(* IEC 61131-3 sources: sphere-usecases/sector-water/rovisys-distribution/implementations/openplc/st, 2 files *)

(* ---- wd_controller.st ---- *)
(*
 * Water Distribution UC0 Controller
 * SPHERE CPS Enclave - OpenPLC Implementation
 *
 * IEC 61131-3 Structured Text (OpenPLC/matiec compatible)
 *
 * This controller manages:
 *   - Supply Line: Supply tank level control, pump operation
 *   - Distribution Grid: Elevated tank filling via valve control
 *   - Return Water System: RWS tank level control, pump operation
 *
 * Architecture:
 *   Controller PLC <-> Modbus Bridge <-> Simulator PLC
 *
 * I/O Mapping (configured in OpenPLC web interface):
 *   Inputs from Simulator (via Bridge):
 *     ai_supply_tank_level -> %IW70
 *     ai_supply_pump_flow -> %IW71
 *     ai_supply_naocl_level -> %IW72
 *     ai_supply_nh4cl_level -> %IW73
 *     ai_grid_elev_level -> %IW74
 *     ai_grid_consum_level -> %IW75
 *     ai_rws_tank_level -> %IW76
 *     di_supply_pump_sts -> %IX2.0
 *     di_supply_mixer_sts -> %IX2.1
 *     di_supply_valve_sts -> %IX2.2
 *     di_grid_elev_valve_sts -> %IX2.3
 *     di_rws_pump_sts -> %IX2.4
 *     di_rws_valve_sts -> %IX2.5
 *     hmi_start -> %IX0.0
 *     hmi_stop -> %IX0.1
 *
 *   Outputs to Simulator (via Bridge):
 *     ao_supply_pump_speed -> %QW100
 *     ao_rws_pump_speed -> %QW101
 *     do_supply_valve -> %QX5.0
 *     do_grid_elev_valve -> %QX5.1
 *     do_rws_valve -> %QX5.2
 *     do_sys_idle -> %QX7.0
 *     do_sys_running -> %QX7.1
 *     do_alarm_supply_hh -> %QX8.0
 *)

(* System State Type - Using INT since iec2c doesn't support ENUM well *)
(* 0=IDLE, 1=START, 2=RUNNING, 3=SHUTDOWN *)

PROGRAM MainProgram
  VAR_INPUT
    (* Analog Inputs from Simulator *)
    ai_supply_tank_level : REAL;      (* Supply tank level [mm] *)
    ai_supply_pump_flow : REAL;       (* Supply pump flow [L/min] *)
    ai_supply_naocl_level : REAL;     (* NaOCl tank level [mm] *)
    ai_supply_nh4cl_level : REAL;     (* NH4Cl tank level [mm] *)
    ai_grid_elev_level : REAL;        (* Elevated tank level [mm] *)
    ai_grid_consum_level : REAL;      (* Consumer tank level [mm] *)
    ai_rws_tank_level : REAL;         (* RWS tank level [mm] *)

    (* Digital Inputs from Simulator *)
    di_supply_pump_sts : BOOL;        (* Supply pump running *)
    di_supply_mixer_sts : BOOL;       (* Supply mixer running *)
    di_supply_valve_sts : BOOL;       (* Supply valve open *)
    di_grid_elev_valve_sts : BOOL;    (* Elevated tank valve open *)
    di_rws_pump_sts : BOOL;           (* RWS pump running *)
    di_rws_valve_sts : BOOL;          (* RWS valve open *)

    (* HMI Inputs *)
    hmi_start : BOOL;                 (* Start button *)
    hmi_stop : BOOL;                  (* Stop button *)
  END_VAR

  VAR_OUTPUT
    (* Analog Outputs to Simulator *)
    ao_supply_pump_speed : REAL;      (* Supply pump speed [%] *)
    ao_rws_pump_speed : REAL;         (* RWS pump speed [%] *)

    (* Digital Outputs to Simulator *)
    do_supply_valve : BOOL;           (* Supply valve command *)
    do_grid_elev_valve : BOOL;        (* Elevated tank valve command *)
    do_rws_valve : BOOL;              (* RWS valve command *)

    (* System State Outputs *)
    do_sys_idle : BOOL;               (* System idle state *)
    do_sys_running : BOOL;            (* System running state *)

    (* Alarm Outputs *)
    do_alarm_supply_hh : BOOL;        (* Supply tank HH alarm *)
  END_VAR

  VAR
    (* System State Machine - 0=IDLE, 1=START, 2=RUNNING, 3=SHUTDOWN *)
    sys_state : INT := 0;
    permissive_supply_ok : BOOL := FALSE;
    permissive_grid_ok : BOOL := FALSE;
    permissives_ready : BOOL := FALSE;

    (* Control Setpoints *)
    supply_tank_low_sp : REAL := 500.0;         (* Start pump below this [mm] *)
    supply_tank_high_sp : REAL := 1200.0;       (* Stop pump above this [mm] *)
    supply_tank_hh_sp : REAL := 1200.0;         (* HH alarm threshold [mm] *)

    grid_elev_low_sp : REAL := 600.0;           (* Open valve below this [mm] *)
    grid_elev_high_sp : REAL := 1600.0;         (* Close valve above this [mm] *)

    rws_tank_low_sp : REAL := 300.0;            (* Start pump below this [mm] *)
    rws_tank_high_sp : REAL := 1200.0;          (* Stop pump above this [mm] *)

    (* Pump Speed Setpoints *)
    supply_pump_normal_speed : REAL := 75.0;    (* Normal operating speed [%] *)
    rws_pump_normal_speed : REAL := 50.0;       (* Normal operating speed [%] *)

    (* Internal State *)
    supply_pump_cmd : BOOL := FALSE;
    rws_pump_cmd : BOOL := FALSE;
  END_VAR

  (* State constants *)
  (* STATE_IDLE = 0; STATE_START = 1; STATE_RUNNING = 2; STATE_SHUTDOWN = 3 *)

  CASE sys_state OF

    0: (* STATE_IDLE - System is idle, waiting for start command *)
      do_sys_idle := TRUE;
      do_sys_running := FALSE;

      (* All outputs off in idle *)
      ao_supply_pump_speed := 0.0;
      ao_rws_pump_speed := 0.0;
      do_supply_valve := FALSE;
      do_grid_elev_valve := FALSE;
      do_rws_valve := FALSE;

      (* Transition: Start button pressed *)
      IF hmi_start AND NOT hmi_stop THEN
        sys_state := 1;
      END_IF;

    1: (* STATE_START - Starting up, check permissives *)
      do_sys_idle := FALSE;
      do_sys_running := FALSE;

      (* Check permissives *)
      permissive_supply_ok := (ai_supply_tank_level > 300.0);
      permissive_grid_ok := (ai_grid_elev_level < 5500.0);
      permissives_ready := permissive_supply_ok AND permissive_grid_ok;

      (* Transition: Permissives met -> RUNNING *)
      IF permissives_ready THEN
        sys_state := 2;
      END_IF;

      (* Transition: Stop pressed -> SHUTDOWN *)
      IF hmi_stop THEN
        sys_state := 3;
      END_IF;

    2: (* STATE_RUNNING - Normal operation *)
      do_sys_idle := FALSE;
      do_sys_running := TRUE;

      (* SUPPLY LINE CONTROL *)
      (* Level-based pump control *)
      IF ai_supply_tank_level <= supply_tank_low_sp THEN
        supply_pump_cmd := TRUE;
      ELSIF ai_supply_tank_level >= supply_tank_high_sp THEN
        supply_pump_cmd := FALSE;
      END_IF;

      (* Set pump speed *)
      IF supply_pump_cmd THEN
        ao_supply_pump_speed := supply_pump_normal_speed;
        do_supply_valve := TRUE;
      ELSE
        ao_supply_pump_speed := 0.0;
        do_supply_valve := FALSE;
      END_IF;

      (* Supply tank HH alarm *)
      IF ai_supply_tank_level >= supply_tank_hh_sp THEN
        do_alarm_supply_hh := TRUE;
      ELSE
        do_alarm_supply_hh := FALSE;
      END_IF;

      (* DISTRIBUTION GRID CONTROL *)
      IF ai_grid_elev_level <= grid_elev_low_sp THEN
        do_grid_elev_valve := TRUE;
      ELSIF ai_grid_elev_level >= grid_elev_high_sp THEN
        do_grid_elev_valve := FALSE;
      END_IF;

      (* RETURN WATER SYSTEM CONTROL *)
      IF ai_rws_tank_level >= rws_tank_high_sp THEN
        rws_pump_cmd := TRUE;
      ELSIF ai_rws_tank_level <= rws_tank_low_sp THEN
        rws_pump_cmd := FALSE;
      END_IF;

      IF rws_pump_cmd THEN
        ao_rws_pump_speed := rws_pump_normal_speed;
        do_rws_valve := TRUE;
      ELSE
        ao_rws_pump_speed := 0.0;
        do_rws_valve := FALSE;
      END_IF;

      (* Transition: Stop pressed -> SHUTDOWN *)
      IF hmi_stop THEN
        sys_state := 3;
      END_IF;

    3: (* STATE_SHUTDOWN - Shutting down *)
      do_sys_idle := FALSE;
      do_sys_running := FALSE;

      (* Stop all pumps *)
      ao_supply_pump_speed := 0.0;
      ao_rws_pump_speed := 0.0;
      supply_pump_cmd := FALSE;
      rws_pump_cmd := FALSE;

      (* Close all valves *)
      do_supply_valve := FALSE;
      do_grid_elev_valve := FALSE;
      do_rws_valve := FALSE;

      (* Clear alarms *)
      do_alarm_supply_hh := FALSE;

      (* Clear permissives *)
      permissive_supply_ok := FALSE;
      permissive_grid_ok := FALSE;
      permissives_ready := FALSE;

      (* Transition: Stop released -> IDLE *)
      IF NOT hmi_stop THEN
        sys_state := 0;
      END_IF;

  END_CASE;

END_PROGRAM

(* ---- wd_simulator.st ---- *)
(*
 * Water Distribution UC0 Simulator
 * SPHERE CPS Enclave - OpenPLC Implementation
 *
 * IEC 61131-3 Structured Text (OpenPLC/matiec compatible)
 *
 * This simulator models the physical dynamics of:
 *   - Supply Line: Supply tank, chemical tanks, pump, valves
 *   - Distribution Grid: Elevated tank, consumer tank, valves
 *   - Return Water System: RWS tank, pump, valves
 *
 * Architecture:
 *   Controller PLC <-> Modbus Bridge <-> Simulator PLC (this)
 *
 * I/O Mapping (configured in OpenPLC web interface):
 *   Command Inputs (from Controller via Bridge):
 *     cmd_supply_pump_speed -> %QW200
 *     cmd_rws_pump_speed -> %QW201
 *     cmd_supply_valve -> %QX3.0
 *     cmd_grid_elev_valve -> %QX3.1
 *     cmd_rws_valve -> %QX3.2
 *
 *   Sensor Outputs (to Controller via Bridge):
 *     out_supply_tank_level -> %QW300
 *     out_supply_pump_flow -> %QW301
 *     out_supply_naocl_level -> %QW302
 *     out_supply_nh4cl_level -> %QW303
 *     out_grid_elev_level -> %QW304
 *     out_grid_consum_level -> %QW305
 *     out_rws_tank_level -> %QW306
 *
 *   Status Outputs (to Controller via Bridge):
 *     out_supply_pump_sts -> %QX40.0
 *     out_supply_mixer_sts -> %QX40.1
 *     out_supply_valve_sts -> %QX40.2
 *     out_grid_elev_valve_sts -> %QX40.3
 *     out_rws_pump_sts -> %QX40.4
 *     out_rws_valve_sts -> %QX40.5
 *)

PROGRAM MainProgram
  VAR_INPUT
    (* Command Inputs from Controller via Bridge *)
    cmd_supply_pump_speed : REAL;     (* Supply pump speed cmd [%] *)
    cmd_rws_pump_speed : REAL;        (* RWS pump speed cmd [%] *)
    cmd_supply_valve : BOOL;          (* Supply valve command *)
    cmd_grid_elev_valve : BOOL;       (* Elevated tank valve cmd *)
    cmd_rws_valve : BOOL;             (* RWS valve command *)
  END_VAR

  VAR_OUTPUT
    (* Sensor Outputs to Controller via Bridge *)
    out_supply_tank_level : REAL;     (* Supply tank level [mm] *)
    out_supply_pump_flow : REAL;      (* Supply pump flow [L/min] *)
    out_supply_naocl_level : REAL;    (* NaOCl tank level [mm] *)
    out_supply_nh4cl_level : REAL;    (* NH4Cl tank level [mm] *)
    out_grid_elev_level : REAL;       (* Elevated tank level [mm] *)
    out_grid_consum_level : REAL;     (* Consumer tank level [mm] *)
    out_rws_tank_level : REAL;        (* RWS tank level [mm] *)

    (* Status Outputs to Controller via Bridge *)
    out_supply_pump_sts : BOOL;       (* Supply pump running *)
    out_supply_mixer_sts : BOOL;      (* Supply mixer running *)
    out_supply_valve_sts : BOOL;      (* Supply valve open *)
    out_grid_elev_valve_sts : BOOL;   (* Elevated tank valve open *)
    out_rws_pump_sts : BOOL;          (* RWS pump running *)
    out_rws_valve_sts : BOOL;         (* RWS valve open *)
  END_VAR

  VAR
    (* Simulation Constants - Timing *)
    DT_SEC : REAL := 0.1;                       (* Simulation timestep [s] *)
    MOTORIZED_VALVE_DELAY : INT := 600;         (* 60s at 100ms scan *)
    PUMP_SPINUP_DELAY : INT := 20;              (* 2s at 100ms scan *)

    (* Physical parameters - Supply *)
    SUPPLY_TANK_AREA_M2 : REAL := 40.0;
    SUPPLY_TANK_MAX_MM : REAL := 1500.0;
    SUPPLY_INFLOW_LPM : REAL := 150.0;
    SUPPLY_PUMP_MAX_LPM : REAL := 200.0;

    (* Physical parameters - Chemical tanks *)
    NAOCL_TANK_AREA_M2 : REAL := 0.1;
    NAOCL_DOSE_LPM : REAL := 0.038;
    NH4CL_TANK_AREA_M2 : REAL := 0.1;
    NH4CL_DOSE_LPM : REAL := 0.019;

    (* Physical parameters - Grid *)
    ELEV_TANK_AREA_M2 : REAL := 60.0;
    ELEV_TANK_MAX_MM : REAL := 2000.0;
    CONSUM_TANK_AREA_M2 : REAL := 10.0;
    CONSUM_TANK_MAX_MM : REAL := 2000.0;
    GRID_DEMAND_LPM : REAL := 100.0;
    ELEV_DRAIN_LPM : REAL := 300.0;

    (* Physical parameters - RWS *)
    RWS_TANK_AREA_M2 : REAL := 0.3;
    RWS_TANK_MAX_MM : REAL := 1500.0;
    RWS_PUMP_MAX_LPM : REAL := 38.0;
    RETURN_FRACTION : REAL := 0.9;

    (* Tank levels [mm] *)
    supply_tank_level : REAL := 1000.0;
    naocl_tank_level : REAL := 800.0;
    nh4cl_tank_level : REAL := 800.0;
    grid_elev_level : REAL := 1200.0;
    grid_consum_level : REAL := 1000.0;
    rws_tank_level : REAL := 500.0;

    (* Valve states with delay modeling *)
    supply_valve_timer : INT := 0;
    supply_valve_state : BOOL := FALSE;
    grid_elev_valve_timer : INT := 0;
    grid_elev_valve_state : BOOL := FALSE;
    rws_valve_timer : INT := 0;
    rws_valve_state : BOOL := FALSE;

    (* Pump states with delay modeling *)
    supply_pump_timer : INT := 0;
    supply_pump_state : BOOL := FALSE;
    supply_pump_actual_speed : REAL := 0.0;
    rws_pump_timer : INT := 0;
    rws_pump_state : BOOL := FALSE;
    rws_pump_actual_speed : REAL := 0.0;

    (* Flow rates [L/min] *)
    supply_pump_flow : REAL := 0.0;
    rws_pump_flow : REAL := 0.0;
    grid_demand_actual : REAL := 0.0;
    return_flow : REAL := 0.0;

    (* Mixer state *)
    mixer_running : BOOL := TRUE;

    (* Temporary calculation variables *)
    delta_level : REAL := 0.0;
    flow_in : REAL := 0.0;
    flow_out : REAL := 0.0;
  END_VAR

  (* =====================================================================
     VALVE DELAY MODELING
     ===================================================================== *)

  (* Supply Tank Valve *)
  IF cmd_supply_valve AND NOT supply_valve_state THEN
    supply_valve_timer := supply_valve_timer + 1;
    IF supply_valve_timer >= MOTORIZED_VALVE_DELAY THEN
      supply_valve_state := TRUE;
      supply_valve_timer := MOTORIZED_VALVE_DELAY;
    END_IF;
  ELSIF NOT cmd_supply_valve AND supply_valve_state THEN
    supply_valve_timer := supply_valve_timer - 1;
    IF supply_valve_timer <= 0 THEN
      supply_valve_state := FALSE;
      supply_valve_timer := 0;
    END_IF;
  ELSIF cmd_supply_valve AND supply_valve_state THEN
    supply_valve_timer := MOTORIZED_VALVE_DELAY;
  ELSE
    supply_valve_timer := 0;
  END_IF;

  (* Grid Elevated Tank Valve *)
  IF cmd_grid_elev_valve AND NOT grid_elev_valve_state THEN
    grid_elev_valve_timer := grid_elev_valve_timer + 1;
    IF grid_elev_valve_timer >= MOTORIZED_VALVE_DELAY THEN
      grid_elev_valve_state := TRUE;
      grid_elev_valve_timer := MOTORIZED_VALVE_DELAY;
    END_IF;
  ELSIF NOT cmd_grid_elev_valve AND grid_elev_valve_state THEN
    grid_elev_valve_timer := grid_elev_valve_timer - 1;
    IF grid_elev_valve_timer <= 0 THEN
      grid_elev_valve_state := FALSE;
      grid_elev_valve_timer := 0;
    END_IF;
  ELSIF cmd_grid_elev_valve AND grid_elev_valve_state THEN
    grid_elev_valve_timer := MOTORIZED_VALVE_DELAY;
  ELSE
    grid_elev_valve_timer := 0;
  END_IF;

  (* RWS Tank Valve *)
  IF cmd_rws_valve AND NOT rws_valve_state THEN
    rws_valve_timer := rws_valve_timer + 1;
    IF rws_valve_timer >= MOTORIZED_VALVE_DELAY THEN
      rws_valve_state := TRUE;
      rws_valve_timer := MOTORIZED_VALVE_DELAY;
    END_IF;
  ELSIF NOT cmd_rws_valve AND rws_valve_state THEN
    rws_valve_timer := rws_valve_timer - 1;
    IF rws_valve_timer <= 0 THEN
      rws_valve_state := FALSE;
      rws_valve_timer := 0;
    END_IF;
  ELSIF cmd_rws_valve AND rws_valve_state THEN
    rws_valve_timer := MOTORIZED_VALVE_DELAY;
  ELSE
    rws_valve_timer := 0;
  END_IF;

  (* =====================================================================
     PUMP DELAY MODELING
     ===================================================================== *)

  (* Supply Pump *)
  IF cmd_supply_pump_speed > 0.0 THEN
    IF NOT supply_pump_state THEN
      supply_pump_timer := supply_pump_timer + 1;
      IF supply_pump_timer >= PUMP_SPINUP_DELAY THEN
        supply_pump_state := TRUE;
      END_IF;
    END_IF;
    IF supply_pump_state THEN
      IF supply_pump_actual_speed < cmd_supply_pump_speed THEN
        supply_pump_actual_speed := supply_pump_actual_speed + 1.0;
        IF supply_pump_actual_speed > cmd_supply_pump_speed THEN
          supply_pump_actual_speed := cmd_supply_pump_speed;
        END_IF;
      ELSIF supply_pump_actual_speed > cmd_supply_pump_speed THEN
        supply_pump_actual_speed := supply_pump_actual_speed - 1.0;
        IF supply_pump_actual_speed < cmd_supply_pump_speed THEN
          supply_pump_actual_speed := cmd_supply_pump_speed;
        END_IF;
      END_IF;
    END_IF;
  ELSE
    supply_pump_timer := 0;
    supply_pump_state := FALSE;
    supply_pump_actual_speed := 0.0;
  END_IF;

  (* RWS Pump *)
  IF cmd_rws_pump_speed > 0.0 THEN
    IF NOT rws_pump_state THEN
      rws_pump_timer := rws_pump_timer + 1;
      IF rws_pump_timer >= PUMP_SPINUP_DELAY THEN
        rws_pump_state := TRUE;
      END_IF;
    END_IF;
    IF rws_pump_state THEN
      IF rws_pump_actual_speed < cmd_rws_pump_speed THEN
        rws_pump_actual_speed := rws_pump_actual_speed + 1.0;
        IF rws_pump_actual_speed > cmd_rws_pump_speed THEN
          rws_pump_actual_speed := cmd_rws_pump_speed;
        END_IF;
      ELSIF rws_pump_actual_speed > cmd_rws_pump_speed THEN
        rws_pump_actual_speed := rws_pump_actual_speed - 1.0;
        IF rws_pump_actual_speed < cmd_rws_pump_speed THEN
          rws_pump_actual_speed := cmd_rws_pump_speed;
        END_IF;
      END_IF;
    END_IF;
  ELSE
    rws_pump_timer := 0;
    rws_pump_state := FALSE;
    rws_pump_actual_speed := 0.0;
  END_IF;

  (* =====================================================================
     FLOW CALCULATIONS
     ===================================================================== *)

  IF supply_pump_state AND supply_valve_state THEN
    supply_pump_flow := (supply_pump_actual_speed / 100.0) * SUPPLY_PUMP_MAX_LPM;
  ELSE
    supply_pump_flow := 0.0;
  END_IF;

  IF rws_pump_state AND rws_valve_state THEN
    rws_pump_flow := (rws_pump_actual_speed / 100.0) * RWS_PUMP_MAX_LPM;
  ELSE
    rws_pump_flow := 0.0;
  END_IF;

  grid_demand_actual := GRID_DEMAND_LPM;
  return_flow := grid_demand_actual * RETURN_FRACTION;

  (* =====================================================================
     MASS BALANCE CALCULATIONS
     ===================================================================== *)

  (* Supply Tank Mass Balance *)
  flow_in := SUPPLY_INFLOW_LPM + rws_pump_flow;
  flow_out := supply_pump_flow;
  delta_level := ((flow_in - flow_out) / SUPPLY_TANK_AREA_M2) * DT_SEC / 60.0 * 1000.0;
  supply_tank_level := supply_tank_level + delta_level;

  IF supply_tank_level < 0.0 THEN
    supply_tank_level := 0.0;
  ELSIF supply_tank_level > SUPPLY_TANK_MAX_MM THEN
    supply_tank_level := SUPPLY_TANK_MAX_MM;
  END_IF;

  (* Chemical Tank Drain *)
  IF supply_pump_state THEN
    delta_level := (NAOCL_DOSE_LPM / NAOCL_TANK_AREA_M2) * DT_SEC / 60.0 * 1000.0;
    naocl_tank_level := naocl_tank_level - delta_level;
    IF naocl_tank_level < 0.0 THEN
      naocl_tank_level := 0.0;
    END_IF;

    delta_level := (NH4CL_DOSE_LPM / NH4CL_TANK_AREA_M2) * DT_SEC / 60.0 * 1000.0;
    nh4cl_tank_level := nh4cl_tank_level - delta_level;
    IF nh4cl_tank_level < 0.0 THEN
      nh4cl_tank_level := 0.0;
    END_IF;
  END_IF;

  (* Elevated Tank Mass Balance *)
  IF grid_elev_valve_state THEN
    flow_in := supply_pump_flow;
  ELSE
    flow_in := 0.0;
  END_IF;
  flow_out := ELEV_DRAIN_LPM;
  delta_level := ((flow_in - flow_out) / ELEV_TANK_AREA_M2) * DT_SEC / 60.0 * 1000.0;
  grid_elev_level := grid_elev_level + delta_level;

  IF grid_elev_level < 0.0 THEN
    grid_elev_level := 0.0;
  ELSIF grid_elev_level > ELEV_TANK_MAX_MM THEN
    grid_elev_level := ELEV_TANK_MAX_MM;
  END_IF;

  (* Consumer Tank Mass Balance *)
  flow_in := ELEV_DRAIN_LPM;
  flow_out := grid_demand_actual;
  delta_level := ((flow_in - flow_out) / CONSUM_TANK_AREA_M2) * DT_SEC / 60.0 * 1000.0;
  grid_consum_level := grid_consum_level + delta_level;

  IF grid_consum_level < 0.0 THEN
    grid_consum_level := 0.0;
  ELSIF grid_consum_level > CONSUM_TANK_MAX_MM THEN
    grid_consum_level := CONSUM_TANK_MAX_MM;
  END_IF;

  (* RWS Tank Mass Balance *)
  flow_in := return_flow;
  flow_out := rws_pump_flow;
  delta_level := ((flow_in - flow_out) / RWS_TANK_AREA_M2) * DT_SEC / 60.0 * 1000.0;
  rws_tank_level := rws_tank_level + delta_level;

  IF rws_tank_level < 0.0 THEN
    rws_tank_level := 0.0;
  ELSIF rws_tank_level > RWS_TANK_MAX_MM THEN
    rws_tank_level := RWS_TANK_MAX_MM;
  END_IF;

  (* =====================================================================
     OUTPUT UPDATES
     ===================================================================== *)

  out_supply_tank_level := supply_tank_level;
  out_supply_pump_flow := supply_pump_flow;
  out_supply_naocl_level := naocl_tank_level;
  out_supply_nh4cl_level := nh4cl_tank_level;
  out_grid_elev_level := grid_elev_level;
  out_grid_consum_level := grid_consum_level;
  out_rws_tank_level := rws_tank_level;

  out_supply_pump_sts := supply_pump_state;
  out_supply_mixer_sts := mixer_running;
  out_supply_valve_sts := supply_valve_state;
  out_grid_elev_valve_sts := grid_elev_valve_state;
  out_rws_pump_sts := rws_pump_state;
  out_rws_valve_sts := rws_valve_state;

END_PROGRAM
